{attribute addProperty BoxType "EL5021-0000-0016"}
{attribute addProperty Id "ENC_StatusAT %I*ENC_Status_33FDC79E80100ENC_ControlAT %Q*ENC_Control_2DBD69A94860WcStateAT %I*WcState_98A4DF7520.250InfoDataAT %I*InfoData_BC63D37F80100"}
{attribute addProperty CRC "2553768403"}
{attribute addProperty SizeInBites "210"}
{attribute addProperty SizeInBytes "26.25"}
TYPE EL5021_32D1A2A3 :
STRUCT
	{attribute addProperty Name "ENC_Status"}
	ENC_Status : ENC_Status_33FDC79E;
	{attribute addProperty Name "ENC_Control"}
	ENC_Control : ENC_Control_2DBD69A9;
	{attribute addProperty Name "WcState"}
	WcState : WcState_98A4DF75;
	{attribute addProperty Name "InfoData"}
	InfoData : InfoData_BC63D37F;
END_STRUCT
END_TYPE

(* stored: Version 1.2.0.0, ProductVersion 3.1.4024.9
   DUT EL5021_32D1A2A3: Id {42602ae6-9cab-4482-8e73-33e6f899a36e} *)
